(* IEC 61131-3 sources: SHU_NSTV/src/lib/ShutterLib, 4 files *)

(* ---- Shutter.st ---- *)
FUNCTION_BLOCK Shutter IMPLEMENTS BasicControl_OpenClose
VAR_INPUT
END_VAR
VAR_OUTPUT
END_VAR
VAR
	OpenMechanism : ShutterOpenMechanism;
	CloseMechanism : ShutterCloseMechanism;
END_VAR

METHOD Close
    CloseMechanism.Set_Power(TRUE);	// Включаем механизм закрытия
    OpenMechanism.Set_Power(FALSE);	// Выключаем механизм открытия
END_METHOD

METHOD Open
    OpenMechanism.Set_Power(TRUE);	// Включаем механизм открытия
    CloseMechanism.Set_Power(FALSE);	// Выключаем механизм закрытия
END_METHOD

METHOD Stop
    OpenMechanism.Set_Power(FALSE);	// Выключаем механизм открытия
    CloseMechanism.Set_Power(FALSE);	// Выключаем механизм закрытия
END_METHOD
END_FUNCTION_BLOCK

(* ---- Shutter_Control.st ---- *)
FUNCTION_BLOCK Shutter_Control
VAR_INPUT
END_VAR
VAR_OUTPUT
END_VAR
VAR
	ConditionOpen, ConditionClose, ConditionStop : BOOL;
END_VAR

METHOD Close
    VAR_INPUT
        access : BOOL;					// Доступ к функциональному блоку
        device : BasicControl_OpenClose;	// Устройство управления закрытием шторки
    END_VAR
    IF access AND ConditionClose THEN
        device.Close();                // Вызываем метод закрытия затвора
    END_IF
END_METHOD

METHOD Open
    VAR_INPUT
        access : BOOL;					// Доступ к функциональному блоку
        device : BasicControl_OpenClose;	// Устройство управления открытием шторки
    END_VAR
    IF access AND ConditionOpen THEN
        device.Open();                 // Вызываем метод открытия затвора
    END_IF
END_METHOD

METHOD Stop
    VAR_INPUT
        access : BOOL;					// Доступ к функциональному блоку
        device : BasicControl_OpenClose;	// Устройство управления остановкой шторки
    END_VAR
    IF access AND ConditionStop THEN
        device.Stop();                 // Вызываем метод остановки затвора
    END_IF
END_METHOD

PROPERTY AccessToOpen : BOOL
    SET
        ConditionOpen := AccessToOpen;	// Устанавливаем условие открытия шторки
    END_SET
END_PROPERTY

PROPERTY AccessToClose : BOOL
    SET
        ConditionClose := AccessToClose;	// Устанавливаем условие закрытия шторки
    END_SET
END_PROPERTY

PROPERTY AccessToStop : BOOL
    SET
        ConditionStop := AccessToStop;	// Устанавливаем условие остановки шторки
    END_SET
END_PROPERTY
END_FUNCTION_BLOCK

(* ---- ShutterCloseMechanism.st ---- *)
FUNCTION_BLOCK ShutterCloseMechanism IMPLEMENTS BasicControl
VAR_INPUT
END_VAR
VAR_OUTPUT
END_VAR
VAR
	qxPower : BOOL;
END_VAR

METHOD Set_Power
    VAR_INPUT
        x : BOOL;				// Вход сигнала питания
    END_VAR
    qxPower := x;				// Присваиваем значение входного сигнала питания к выходному сигналу
END_METHOD

PROPERTY Power : BOOL
    GET
        Power := qxPower;	// Возвращаем значение выходного сигнала питания
    END_GET
END_PROPERTY
END_FUNCTION_BLOCK

(* ---- ShutterOpenMechanism.st ---- *)
FUNCTION_BLOCK ShutterOpenMechanism IMPLEMENTS BasicControl
VAR_INPUT
END_VAR
VAR_OUTPUT
END_VAR
VAR
	qxPower : BOOL;
END_VAR

METHOD Set_Power
    VAR_INPUT
        x : BOOL;				// Вход сигнала питания
    END_VAR
    qxPower := x;				// Присваиваем значение входного сигнала питания к выходному сигналу
END_METHOD

PROPERTY Power : BOOL
    GET
        Power := qxPower;	// Возвращаем значение выходного сигнала питания
    END_GET
END_PROPERTY
END_FUNCTION_BLOCK
